{attribute 'qualified_only'}
{attribute 'strict'}
{attribute 'to_string'}
TYPE E_ScrewdriverStep :
(
    Idle                       := 0,

    // 首次初始化
    InitializeSafeZ            := 10,
    InitializeYZero            := 20,

    // 预拧紧与避让
    MoveYForPreTighten         := 30,
    LowerForPreTighten         := 40,
    WaitPreTighten             := 50,
    LiftAfterPreTighten        := 60,
    RetreatYToSafe             := 70,

    // Adjustment保持在工作位期间等待业务请求
    WaitProcessRequest         := 80,

    // 二次拧紧
    MoveYForSecondTighten      := 110,
    LowerForSecondTighten      := 120,
    WaitSecondTighten          := 130,
    LiftAfterSecondTighten     := 140,
    RetreatYAfterSecondTighten := 145,
    WaitSecondTightenAck       := 150,

    // 二次拧紧后不合格时的返工拧松
    MoveYForReworkLoosen       := 155,
    LowerForReworkLoosen       := 160,
    WaitReworkLoosen           := 165,
    LiftAfterReworkLoosen      := 170,
    RetreatYAfterReworkLoosen  := 175,
    WaitReworkLoosenAck        := 180,

    // 本机构流程完成后等待周期确认
    WaitDoneAck                := 190,

    Error                      := 900
);
END_TYPE

(* stored: Version 1.1.0.1, ProductVersion 3.1.4026.20
   DUT E_ScrewdriverStep: Id {606c08a8-6dbd-49dc-b77b-aa909f9a5086} *)
